{attribute 'hide'}
FUNCTION F_HwGetAddrInfo_29bit_CX2500_M510 : ST_CanHeader
VAR_INPUT
	stInput: ST_CanData_29bit_CX2500_M510;
END_VAR

F_HwGetAddrInfo_29bit_CX2500_M510.nCobid := 16#3FFFFFFF AND UDINT_TO_DWORD(stInput.nCobid);// limits cobid to max value

F_HwGetAddrInfo_29bit_CX2500_M510.bRTR := stInput.nCobid.30;// gets RTR bit

F_HwGetAddrInfo_29bit_CX2500_M510.bExtendedAddress := stInput.nCobid.31;//gets extended address flag, if set raw can message had 29bit for identification on the wire.

IF (stInput.nLength > 8) THEN
	F_HwGetAddrInfo_29bit_CX2500_M510.nMsgLength := 8;
ELSE
	F_HwGetAddrInfo_29bit_CX2500_M510.nMsgLength := stInput.nLength;
END_IF

END_FUNCTION

(* stored: Version 1.1.0.1, ProductVersion 3.1.4024.12
   POU F_HwGetAddrInfo_29bit_CX2500_M510: Id {b5a7888b-4d98-08b0-1922-0059968f8013}, SpecialFunc None *)
